FUNCTION TryConvert_BOOL_TO_BOOL : BOOL
VAR_INPUT
	in : BOOL;
	out : REFERENCE TO BOOL;
END_VAR

out := in;
TryConvert_BOOL_TO_BOOL := TRUE;

END_FUNCTION

(* stored: Version 1.1.0.1, ProductVersion 3.1.4024.12
   POU TryConvert_BOOL_TO_BOOL: Id {a09228d4-d045-4367-a06e-22827c2785f8}, SpecialFunc None *)
